// Mitsubishi GX Developer project: PLC-3floor-elevator   PLC: FX2N

PROGRAM MAIN
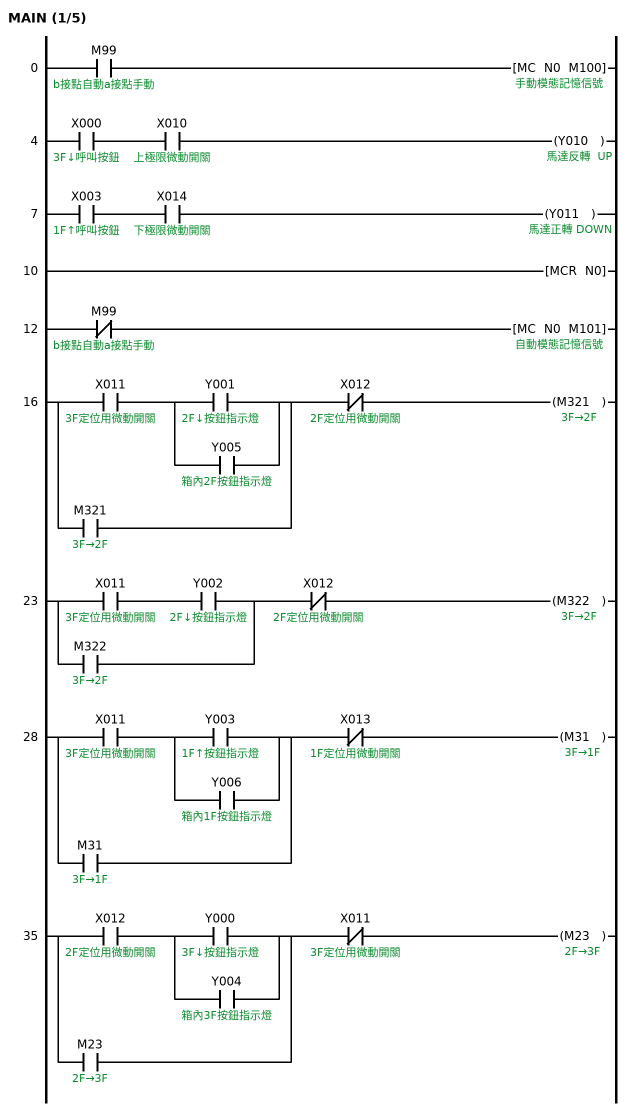
0     LD      M99  ; b接點自動a接點手動
      MC      N0 M100  ; 手動模態記憶信號
4     LD      X000  ; 3F↓呼叫按鈕
      AND     X010  ; 上極限微動開關
      OUT     Y010  ; 馬達反轉  UP
7     LD      X003  ; 1F↑呼叫按鈕
      AND     X014  ; 下極限微動開關
      OUT     Y011  ; 馬達正轉 DOWN
10    MCR     N0
12    LDI     M99  ; b接點自動a接點手動
      MC      N0 M101  ; 自動模態記憶信號
16    LD      X011  ; 3F定位用微動開關
      LD      Y001  ; 2F↓按鈕指示燈
      OR      Y005  ; 箱內2F按鈕指示燈
      ANB
      OR      M321  ; 3F→2F
      ANI     X012  ; 2F定位用微動開關
      OUT     M321  ; 3F→2F
23    LD      X011  ; 3F定位用微動開關
      AND     Y002  ; 2F↓按鈕指示燈
      OR      M322  ; 3F→2F
      ANI     X012  ; 2F定位用微動開關
      OUT     M322  ; 3F→2F
28    LD      X011  ; 3F定位用微動開關
      LD      Y003  ; 1F↑按鈕指示燈
      OR      Y006  ; 箱內1F按鈕指示燈
      ANB
      OR      M31  ; 3F→1F
      ANI     X013  ; 1F定位用微動開關
      OUT     M31  ; 3F→1F
35    LD      X012  ; 2F定位用微動開關
      LD      Y000  ; 3F↓按鈕指示燈
      OR      Y004  ; 箱內3F按鈕指示燈
      ANB
      OR      M23  ; 2F→3F
      ANI     X011  ; 3F定位用微動開關
      OUT     M23  ; 2F→3F
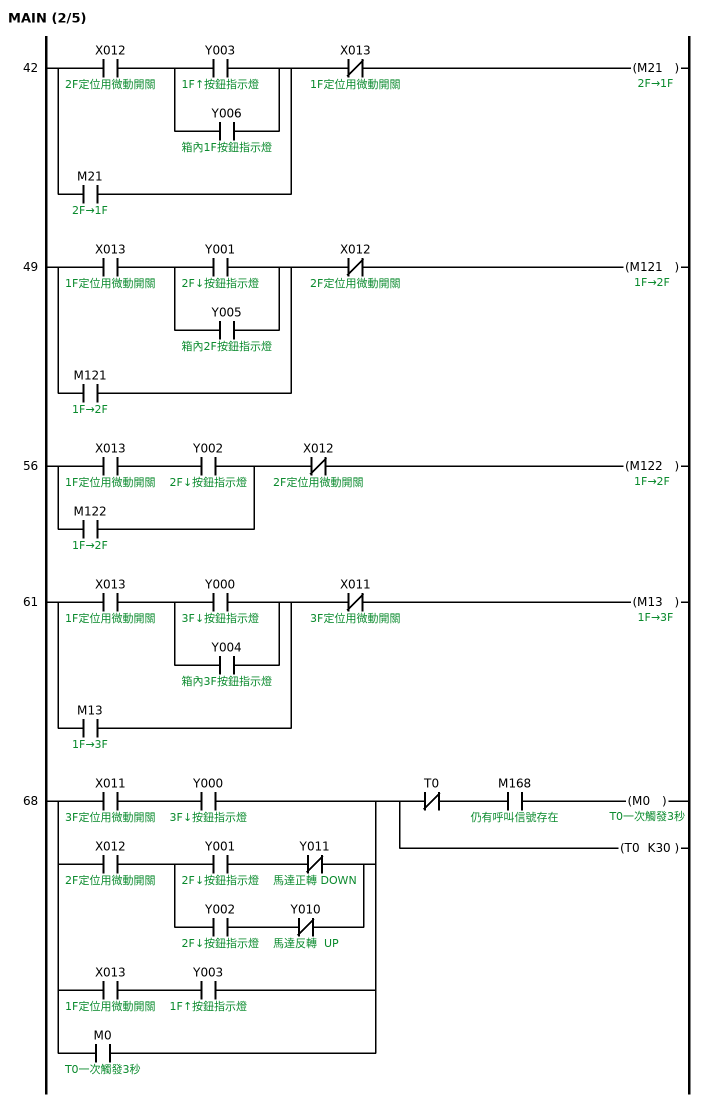
42    LD      X012  ; 2F定位用微動開關
      LD      Y003  ; 1F↑按鈕指示燈
      OR      Y006  ; 箱內1F按鈕指示燈
      ANB
      OR      M21  ; 2F→1F
      ANI     X013  ; 1F定位用微動開關
      OUT     M21  ; 2F→1F
49    LD      X013  ; 1F定位用微動開關
      LD      Y001  ; 2F↓按鈕指示燈
      OR      Y005  ; 箱內2F按鈕指示燈
      ANB
      OR      M121  ; 1F→2F
      ANI     X012  ; 2F定位用微動開關
      OUT     M121  ; 1F→2F
56    LD      X013  ; 1F定位用微動開關
      AND     Y002  ; 2F↓按鈕指示燈
      OR      M122  ; 1F→2F
      ANI     X012  ; 2F定位用微動開關
      OUT     M122  ; 1F→2F
61    LD      X013  ; 1F定位用微動開關
      LD      Y000  ; 3F↓按鈕指示燈
      OR      Y004  ; 箱內3F按鈕指示燈
      ANB
      OR      M13  ; 1F→3F
      ANI     X011  ; 3F定位用微動開關
      OUT     M13  ; 1F→3F
68    LD      X011  ; 3F定位用微動開關
      AND     Y000  ; 3F↓按鈕指示燈
      LD      X012  ; 2F定位用微動開關
      LD      Y001  ; 2F↓按鈕指示燈
      ANI     Y011  ; 馬達正轉 DOWN
      LD      Y002  ; 2F↓按鈕指示燈
      ANI     Y010  ; 馬達反轉  UP
      ORB
      ANB
      ORB
      LD      X013  ; 1F定位用微動開關
      AND     Y003  ; 1F↑按鈕指示燈
      ORB
      OR      M0  ; T0一次觸發3秒
      MPS
      ANI     T0
      AND     M168  ; 仍有呼叫信號存在
      OUT     M0  ; T0一次觸發3秒
      MPP
      OUT     T0 K30
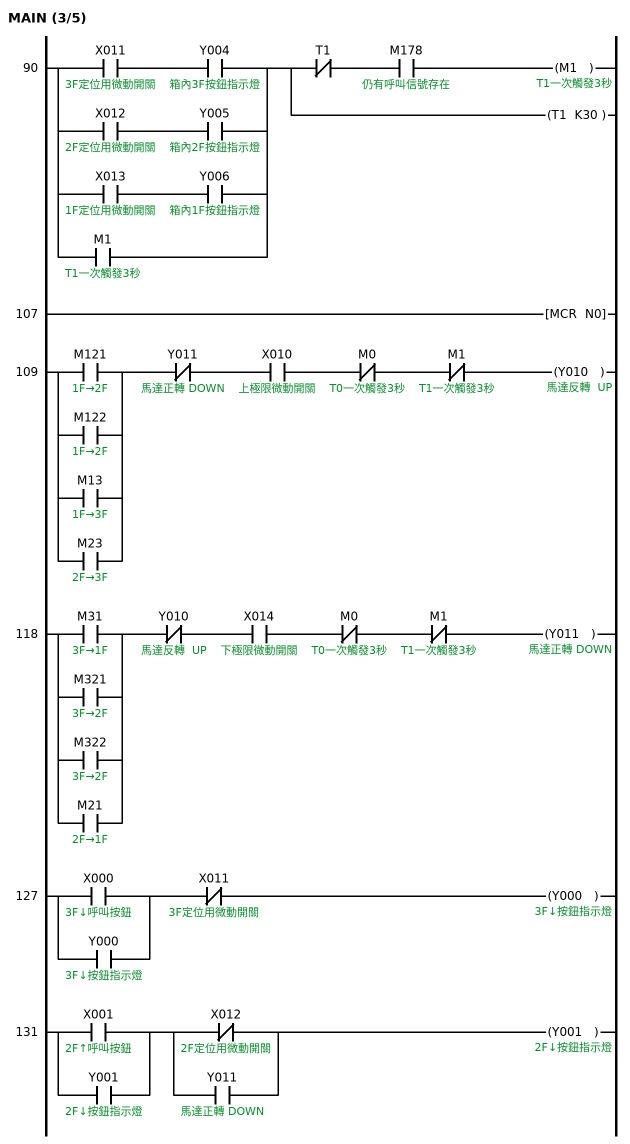
90    LD      X011  ; 3F定位用微動開關
      AND     Y004  ; 箱內3F按鈕指示燈
      LD      X012  ; 2F定位用微動開關
      AND     Y005  ; 箱內2F按鈕指示燈
      ORB
      LD      X013  ; 1F定位用微動開關
      AND     Y006  ; 箱內1F按鈕指示燈
      ORB
      OR      M1  ; T1一次觸發3秒
      MPS
      ANI     T1
      AND     M178  ; 仍有呼叫信號存在
      OUT     M1  ; T1一次觸發3秒
      MPP
      OUT     T1 K30
107   MCR     N0
109   LD      M121  ; 1F→2F
      OR      M122  ; 1F→2F
      OR      M13  ; 1F→3F
      OR      M23  ; 2F→3F
      ANI     Y011  ; 馬達正轉 DOWN
      AND     X010  ; 上極限微動開關
      ANI     M0  ; T0一次觸發3秒
      ANI     M1  ; T1一次觸發3秒
      OUT     Y010  ; 馬達反轉  UP
118   LD      M31  ; 3F→1F
      OR      M321  ; 3F→2F
      OR      M322  ; 3F→2F
      OR      M21  ; 2F→1F
      ANI     Y010  ; 馬達反轉  UP
      AND     X014  ; 下極限微動開關
      ANI     M0  ; T0一次觸發3秒
      ANI     M1  ; T1一次觸發3秒
      OUT     Y011  ; 馬達正轉 DOWN
127   LD      X000  ; 3F↓呼叫按鈕
      OR      Y000  ; 3F↓按鈕指示燈
      ANI     X011  ; 3F定位用微動開關
      OUT     Y000  ; 3F↓按鈕指示燈
131   LD      X001  ; 2F↑呼叫按鈕
      OR      Y001  ; 2F↓按鈕指示燈
      LDI     X012  ; 2F定位用微動開關
      OR      Y011  ; 馬達正轉 DOWN
      ANB
      OUT     Y001  ; 2F↓按鈕指示燈
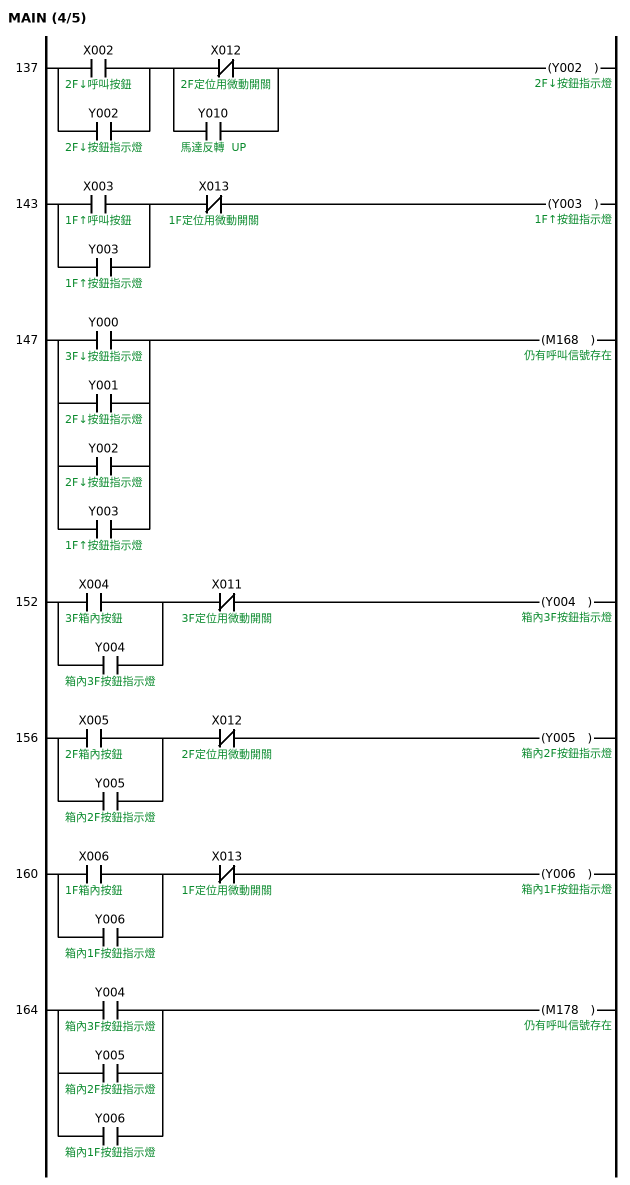
137   LD      X002  ; 2F↓呼叫按鈕
      OR      Y002  ; 2F↓按鈕指示燈
      LDI     X012  ; 2F定位用微動開關
      OR      Y010  ; 馬達反轉  UP
      ANB
      OUT     Y002  ; 2F↓按鈕指示燈
143   LD      X003  ; 1F↑呼叫按鈕
      OR      Y003  ; 1F↑按鈕指示燈
      ANI     X013  ; 1F定位用微動開關
      OUT     Y003  ; 1F↑按鈕指示燈
147   LD      Y000  ; 3F↓按鈕指示燈
      OR      Y001  ; 2F↓按鈕指示燈
      OR      Y002  ; 2F↓按鈕指示燈
      OR      Y003  ; 1F↑按鈕指示燈
      OUT     M168  ; 仍有呼叫信號存在
152   LD      X004  ; 3F箱內按鈕
      OR      Y004  ; 箱內3F按鈕指示燈
      ANI     X011  ; 3F定位用微動開關
      OUT     Y004  ; 箱內3F按鈕指示燈
156   LD      X005  ; 2F箱內按鈕
      OR      Y005  ; 箱內2F按鈕指示燈
      ANI     X012  ; 2F定位用微動開關
      OUT     Y005  ; 箱內2F按鈕指示燈
160   LD      X006  ; 1F箱內按鈕
      OR      Y006  ; 箱內1F按鈕指示燈
      ANI     X013  ; 1F定位用微動開關
      OUT     Y006  ; 箱內1F按鈕指示燈
164   LD      Y004  ; 箱內3F按鈕指示燈
      OR      Y005  ; 箱內2F按鈕指示燈
      OR      Y006  ; 箱內1F按鈕指示燈
      OUT     M178  ; 仍有呼叫信號存在
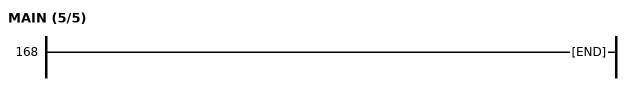
168   END
END_PROGRAM

// device comments not shown above
M12  ; 1F→2F
M32  ; 3F→2F
X007  ; 非常停止按鈕
Y007  ; 非長停止按鈕指示燈
